{attribute addProperty BoxType "EL2911-0000-0016"}
{attribute addProperty Id "FSoE_CommandUSINT811FSOUT_Module_Module_FaultBIT10.1251FSIN_Module_Channel_1_InputBIT10.1251FSIN_Module_Channel_2_InputBIT10.1252FSIN_Module_Channel_3_InputBIT10.1253FSIN_Module_Channel_4_InputBIT10.1254FSIN_Module_Module_FaultBIT10.1251FSoE_CRC_000UINT1623FSoE_Connection_IDUINT1622"}
{attribute addProperty CRC "159468485"}
{attribute addProperty SizeInBites "48"}
{attribute addProperty SizeInBytes "6"}
TYPE FSOE_09814BC5 :
STRUCT
	{attribute addProperty Name "FSoE_Command"}
	FSoE_Command : USINT;
	{attribute addProperty Name "FSOUT_Module_Module_Fault"}
	FSOUT_Module_Module_Fault : BIT;
	{attribute addProperty Name "FSIN_Module_Channel_1_Input"}
	FSIN_Module_Channel_1_Input : BIT;
	{attribute addProperty Name "FSIN_Module_Channel_2_Input"}
	FSIN_Module_Channel_2_Input : BIT;
	{attribute addProperty Name "FSIN_Module_Channel_3_Input"}
	FSIN_Module_Channel_3_Input : BIT;
	{attribute addProperty Name "FSIN_Module_Channel_4_Input"}
	FSIN_Module_Channel_4_Input : BIT;
	{attribute addProperty Name "FSIN_Module_Module_Fault"}
	FSIN_Module_Module_Fault : BIT;
	{attribute 'hide'}
	reserve_1_BIT_0 : BIT;
	{attribute 'hide'}
	reserve_1_BIT_1 : BIT;
	{attribute addProperty Name "FSoE_CRC_000"}
	FSoE_CRC_000 : UINT;
	{attribute addProperty Name "FSoE_Connection_ID"}
	FSoE_Connection_ID : UINT;
END_STRUCT
END_TYPE

(* stored: Version 1.2.0.0, ProductVersion 3.1.4024.9
   DUT FSOE_09814BC5: Id {114d8b43-ae94-4d39-9fbb-11b025e5bfe6} *)
